//==================================================================================================
//							Beckhoff Automation Poland
//								FB_AntiBlinkAlarmFilter
//									20.12.2016
//				Blok służący do wyłączania logowania zdarzeń które pojawiają się zbyt często
// 	v1.0 || TC v 3.1.4020.28 || - pierwsza wersja
//==================================================================================================
FUNCTION_BLOCK FB_AntiBlinkAlarmFilter
VAR_INPUT
	bEvent			: BOOL;		// Status zdarzenia
	tTime			: TIME;		// Zadane okno czasowe
	uiLimit			: UINT;		// Maksymalna liczba zdarzeń jaka może się pojawić w oknie czasowym
END_VAR
VAR_IN_OUT
	bPermission		: BOOL;		// Flaga zezwolenia na logowanie zdarzeń
END_VAR
VAR
	tStartTime		: TIME;		// Zmienna przechowująca czas rozpoczęcia zliczania
	uiActCount		: UINT;		// Aktualna wartość licznika
	rtEdge			: R_TRIG;	// Zbocze narastające
END_VAR

rtEdge(CLK:=bEvent);
IF rtEdge.Q THEN							// Blok podejmuje akcję w przypadku wystapienia zdarzenia
	IF uiActCount = 0 THEN	
		tStartTime		:= TIME();			// W przypadku gdy licznik wynosi zero, zapisywany jest czas rozpoczęcia zliczania
	END_IF
	uiActCount			:= uiActCount + 1;	// Inkrementacja licznika liczby zdarzeń
	IF uiActcount >= uiLimit THEN			// W przypadku gdy liczba zdarzeń osiągnie zadany limit, sprawdzany jest czas w jakim one wystapiły. Jeśli czas jest większy niż dopuszczalny, resetowana jest flaga zezwolenia
		IF TIME() - tStartTime < tTime THEN
			bPermission	:= FALSE;		
		END_IF
		uiActCount 		:= 0;
	END_IF
	IF NOT bPermission THEN
		uiActCount		:= 0;
	END_IF
END_IF;

END_FUNCTION_BLOCK

(* stored: Version 1.1.0.1, ProductVersion 3.1.4022.12
   POU FB_AntiBlinkAlarmFilter: Id {ee86e843-ab76-4901-a36e-d9e2f7a1a2fa}, SpecialFunc None *)
